PROGRAM FAST
VAR
END_VAR

;

END_PROGRAM

(* stored: Version 1.1.0.1, ProductVersion 3.1.4024.9
   POU FAST: Id {9f60d674-6dff-480f-9336-a78c45dbc093}, SpecialFunc None *)
